{attribute 'pack_mode' := '1'}
TYPE ST_1126_Omni_wheels_ref_struct :
	STRUCT
		Steer_angle_reference : REAL;
		Wheel_speed_reference : REAL;
	END_STRUCT
END_TYPE

(* stored: Version 1.1.0.1, ProductVersion 3.1.4026.17
   DUT ST_1126_Omni_wheels_ref_struct: Id {616f44e3-96e3-4b78-a519-71183f162e63} *)
